FUNCTION F_SET_Event : BOOL
VAR_INPUT
	dwID									: DWORD;
	stEventDefinition						: ST_EventDefinition;
	dtActTime								: DT;
END_VAR
VAR
	i										: DINT;
END_VAR

// Przesun elemety tablicy
FOR i := 0 TO GVL_EHS.diNoOfEvents-2 DO
	GVL_EHSP.arrEvent[GVL_EHS.diNoOfEvents-i] := GVL_EHSP.arrEvent[GVL_EHS.diNoOfEvents-i-1];
END_FOR
// Dodaj nowy
GVL_EHSP.arrEvent[1].dwID					:= dwID;
GVL_EHSP.arrEvent[1].dtDateBegin 			:= dtActTime;
GVL_EHSP.arrEvent[1].dtDateEnd	 			:= DT#1970-1-1-0:0:0;
GVL_EHSP.arrEvent[1].dwParam 				:= stEventDefinition.dwParam;
GVL_EHSP.arrEvent[1].dwClass 				:= stEventDefinition.dwClass;

END_FUNCTION

(* stored: Version 1.1.0.1, ProductVersion 3.1.4020.12
   POU F_SET_Event: Id {a76b0465-c660-484f-b14f-1c181bcc4040}, SpecialFunc None *)
